TYPE ST_CoeEntry_INT EXTENDS ST_CoeEntry :
STRUCT
	Value	: INT;
END_STRUCT
END_TYPE

(* stored: Version 1.1.0.1, ProductVersion 3.1.4024.14
   DUT ST_CoeEntry_INT: Id {37a1bc2a-8576-0072-1016-aba83f22bfb6} *)
